// TIA Portal V17 export
// export: Created 2025-03-07T09:24:29.5443759Z, ExportSetting WithDefaults, DisplayName Totally Integrated Automation Portal, DisplayVersion V17 Update 8, DisplayName TIA Portal Openness, DisplayVersion V17 Update 8, DisplayName TIA Portal Version Control Interface, DisplayVersion V17, DisplayName SINAMICS Startdrive Advanced, DisplayVersion V17 SP2, DisplayName SINAMICS Startdrive G110M, G120, G120C, G120D, G120P, G115D, DisplayVersion V17 SP2, DisplayName SINAMICS Startdrive G130, G150, S120, S150, SINAMICS MV, S210, DisplayVersion V17 SP2, DisplayName STEP 7 Professional, DisplayVersion V17 Update 8, DisplayName SINUMERIK ONE STEP 7 Toolbox, DisplayVersion V17 Update 12, DisplayName SINUMERIK 840D sl STEP 7 Toolbox, DisplayVersion V17 Update 12, DisplayName STEP 7 Safety, DisplayVersion V17 Update 6, DisplayName WinCC Advanced, DisplayVersion V17 Update 8
DATA_BLOCK "DB1021_PLC_CNC_DATA"   // DB1021
{ S7_Optimized_Access := 'TRUE'; DB_Accessible_From_OPC_UA := 'FALSE' }
VERSION : 0.1
// stored: AutoNumber false, DBAccessibleFromOPCUA false, DBAccessibleFromWebserver true, IsOnlyStoredInLoadMemory false, IsRetainMemResEnabled false, IsWriteProtectedInAS false, MemoryReserve 100
   VAR
      SENDDP : Struct
         RET_DPRD : Word;   // NON-FAIL-SAFE ERROR CODE RET_VAL OF THE DPRD_DAT INSTRUCTION
         RET_DPWR : Word;   // NON-FAIL-SAFE ERROR CODE RET_VAL OF THE DPWR_DATA INSTRUCTION
         DIAG : Byte;   // NON-FAIL SAFE SERVICE INFORMATION
      END_STRUCT;
      RCVDP : Struct
         RET_DPRD : Word;   // NON-FAIL-SAFE ERROR CODE RET_VAL OF THE DPRD_DAT INSTRUCTION
         RET_DPWR : Word;   // NON-FAIL-SAFE ERROR CODE RET_VAL OF THE DPWR_DATA INSTRUCTION
         DIAG : Byte;   // NON-FAIL SAFE SERVICE INFORMATION
         ACK_REI : Bool;   // ACKNOWLEDGMENT FOR REINTEGRATION OF SEND DATA FOLLOWING COMMUNICAITON ERROR
      END_STRUCT;
   END_VAR
BEGIN
END_DATA_BLOCK
